# EPICS substitutions: NANODAC/nanodacApp/Db/nanodac.substitutions
file nanodac.db
{
pattern {S, ND, NI}
	{BL99:, SE:ND1:, 1}
}
